FUNCTION F_AtomicMassLookup : LREAL
VAR_INPUT
    sMaterialName : T_MaxString;
END_VAR
VAR
    fbAtomicMass : FB_AtomicMass;
END_VAR


fbAtomicMass(
    sName := sMaterialName
);

IF fbAtomicMass.bFound THEN
    F_AtomicMassLookup := fbAtomicMass.fValue;
ELSE
    F_AtomicMassLookup := -1.0;    
END_IF

END_FUNCTION

(* stored: Version 1.1.0.1
   POU F_AtomicMassLookup: Id {d04265c6-a6db-4d14-8510-380c17bf00f7}, SpecialFunc None *)
